{attribute 'hide'}
FUNCTION F_HwSetAddrInfo_11bit : WORD
VAR_INPUT
	stInput: ST_CanHeader;
END_VAR

F_HwSetAddrInfo_11bit := SHL((16#7FF AND DWORD_TO_WORD(stInput.nCobid)),5); //shift cobid from 0-10 to bits 5-16, limits cobid to max value

F_HwSetAddrInfo_11bit.4 := stInput.bRTR;// gets RTR bit

IF (stInput.nMsgLength > 8) THEN// returns the first bits 0-3 which is data length value, checks to make sure length is not greater than max data length (8);
	F_HwSetAddrInfo_11bit := 8;//issue getting data length, set to max.
ELSE
	F_HwSetAddrInfo_11bit :=  F_HwSetAddrInfo_11bit OR UINT_TO_WORD(stInput.nMsgLength);// sets bits 0-3 which is can data length. 
END_IF

//Extended Indentifier isn't used.

END_FUNCTION

(* stored: Version 1.1.0.1, ProductVersion 3.1.4024.11
   POU F_HwSetAddrInfo_11bit: Id {290e3265-1d84-48f1-aefd-bd3b8eec4a28}, SpecialFunc None *)
